% RSLogix 500 project MLO3B JOB 17_BAK128.RSS, saved by version 10.00.00.00 %
PROJECT "MLO3B"    % processor: Bul.1763 MicroLogix 1100 Series B %

PROGRAM FILES
  LAD 2   6 rungs

DATA FILES
  O0 OUTPUT  4 elements
  I1 INPUT  6 elements
  S2 STATUS  66 elements
  B3 BINARY  1 elements
  T4 TIMER  1 elements
  C5 COUNTER  1 elements
  R6 CONTROL  1 elements
  N7 INTEGER  1 elements
  F8 FLOAT  1 elements

LADDER 2
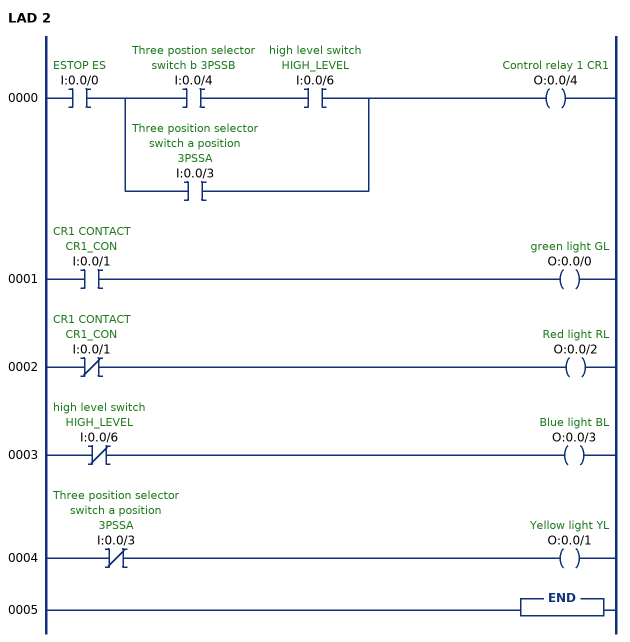
% Rung: 0 %
SOR XIC I:0.0/0 BST XIC I:0.0/4 XIC I:0.0/6 NXB XIC I:0.0/3 BND OTE O:0.0/4 EOR
%   I:0.0/0  ES  "ESTOP" %
%   I:0.0/4  3PSSB  "Three postion selector switch b" %
%   I:0.0/6  HIGH_LEVEL  "high level switch" %
%   I:0.0/3  3PSSA  "Three position selector switch a position" %
%   O:0.0/4  CR1  "Control relay 1" %
% Rung: 1 %
SOR XIC I:0.0/1 OTE O:0.0/0 EOR
%   I:0.0/1  CR1_CON  "CR1 CONTACT" %
%   O:0.0/0  GL  "green light" %
% Rung: 2 %
SOR XIO I:0.0/1 OTE O:0.0/2 EOR
%   I:0.0/1  CR1_CON  "CR1 CONTACT" %
%   O:0.0/2  RL  "Red light" %
% Rung: 3 %
SOR XIO I:0.0/6 OTE O:0.0/3 EOR
%   I:0.0/6  HIGH_LEVEL  "high level switch" %
%   O:0.0/3  BL  "Blue light" %
% Rung: 4 %
SOR XIO I:0.0/3 OTE O:0.0/1 EOR
%   I:0.0/3  3PSSA  "Three position selector switch a position" %
%   O:0.0/1  YL  "Yellow light" %
% Rung: 5 %
SOR END EOR

OTHER DOCUMENTED ADDRESSES
  B3:0/0  CONTACT
  B3:0/1  B  "B CONTACT"
  B3:0/2  "B CONTACT"
  B3:0/3  "b contact"
  B3:0/5  "LAST FWD"
  B3:0/6  "LAST REV"
  B3:0/7  "YELLOW BIT"
  GR  "green light"
  GREE  
  I:0.0/2  CR2C  "CR2 Con"
  I:0.0/5  2PSS  "AUTO/OFF"
  I:0.0/7  PB2  "start"
  I:0.0/8  PB3  "JOG"
  I:0.0/9  LO_LVL  "LOW LEVEL SWITCH"
  I:0.0/10  HIGH_LVL  "HIGH LEVEL SWITCH"
  IOS  
  O:0.0/5  CR2  "Control relay 2"
  O:0.0/6  RED_LIGHT
  O:0.0/7  "Green light"
  T4:0  MOTOR_TIMER  "timer"

COMMENTS NOT ATTACHED TO A CURRENT RUNG
  B3:0/0: FWD-REV using 3 position switch for 1p motor

DATA TABLE (non-zero values as saved)
DATA T4
% .PRE .ACC %
% T4:0 % 8 0
